# EPICS autosave request: measComp/measCompApp/Db/measCompWaveformGenN_settings.req
$(P)$(R)UserWF
$(P)$(R)Enable
$(P)$(R)Type
$(P)$(R)PulseWidth
$(P)$(R)Amplitude
$(P)$(R)Offset
